(* IEC 61131-3 sources: RL_MAR/experiments/comparison/llm4plc/results/deepseek-ai-DeepSeek-V3.2_20260506_104945/20260506_110433, 4 files *)

(* ---- generated_code_iteration_0.st ---- *)
START_ST
FUNCTION_BLOCK ShellSortFB
VAR_INPUT
    sortDirection : BOOL; // FALSE = ascending, TRUE = descending
    arr : ARRAY[1..1000] OF DINT;
END_VAR
VAR_OUTPUT
    error : BOOL;
    status : WORD;
    sorted_arr : ARRAY[1..1000] OF DINT;
END_VAR
VAR
    state : INT; // 0=INIT, 1=SORTING, 2=COMPLETED, 3=ERROR
    prevState : INT;
    i : DINT;
    j : DINT;
    gap : DINT;
    temp : DINT;
    swapFlag : BOOL;
    N : CONSTANT := 1000;
    internalArray : ARRAY[1..1000] OF DINT;
END_VAR

CASE state OF
    0: // STATE 0: INITIALIZE
        // Copy input array to sorted_arr and internalArray
        FOR i := 1 TO N BY 1 DO
            sorted_arr[i] := arr[i];
            internalArray[i] := arr[i];
        END_FOR;

        // Perform array length validation (N is fixed at 1000)
        IF N <= 1 THEN
            error := TRUE;
            status := 16#8200; // Array size <= 1
            state := 3; // Transition to ERROR state
        ELSIF N > 1000 THEN
            error := TRUE;
            status := 16#8201; // Array size > 1000
            state := 3; // Transition to ERROR state
        ELSE
            error := FALSE;
            status := 16#0000; // No error
            state := 1; // Transition to SORTING state
            gap := N / 2; // Initialize gap for Shell Sort
            swapFlag := FALSE;
        END_IF;

    1: // STATE 1: SORTING
        // Perform Shell Sort algorithm
        IF gap > 0 THEN
            swapFlag := FALSE;
            i := gap + 1;
            WHILE i <= N DO
                temp := internalArray[i];
                j := i;

                // Compare and swap based on sortDirection
                IF NOT sortDirection THEN // Ascending order
                    WHILE (j > gap) AND (internalArray[j - gap] > temp) DO
                        internalArray[j] := internalArray[j - gap];
                        j := j - gap;
                        swapFlag := TRUE;
                    END_WHILE;
                ELSE // Descending order
                    WHILE (j > gap) AND (internalArray[j - gap] < temp) DO
                        internalArray[j] := internalArray[j - gap];
                        j := j - gap;
                        swapFlag := TRUE;
                    END_WHILE;
                END_IF;

                internalArray[j] := temp;
                i := i + 1;
            END_WHILE;

            // Reduce gap if no swaps occurred in this iteration
            IF NOT swapFlag THEN
                gap := gap / 2;
            END_IF;
        ELSE
            // Sorting completed, copy internalArray to sorted_arr
            FOR i := 1 TO N BY 1 DO
                sorted_arr[i] := internalArray[i];
            END_FOR;
            state := 2; // Transition to COMPLETED state
        END_IF;

    2: // STATE 2: COMPLETED
        // Maintain final outputs
        error := FALSE;
        status := 16#0000;
        // sorted_arr already contains sorted result
        // Remain in COMPLETED state
        state := 2;

    3: // STATE 3: ERROR
        // Maintain error outputs
        // sorted_arr already contains copy of input arr (unsorted)
        // Remain in ERROR state
        state := 3;

END_CASE;

prevState := state;
END_FUNCTION_BLOCK
END_ST

(* ---- generated_code_iteration_1.st ---- *)
START_REASON
The validation feedback indicates that the CODESYS compiler validation failed with the message: "应该采用类型定义取代'CONSTANT'". This is Chinese for "should use type definition instead of 'CONSTANT'". In CODESYS Structured Text (IEC 61131-3), the keyword for declaring a constant is `CONSTANT`, but the feedback suggests using a type definition. However, `CONSTANT` is the correct keyword for declaring a constant variable within a VAR section. The issue might be that `CONSTANT` is used in a VAR block where it should be declared differently, or there might be a syntax nuance. In CODESYS, constants in a VAR block are declared with `CONSTANT` after the variable name and type, but the feedback might be pointing to using a type definition (e.g., defining a constant at the global scope) instead. Alternatively, the constant `N` is declared as `N : CONSTANT := 1000;` in the VAR section. According to IEC 61131-3, constants in VAR blocks should be declared as `CONSTANT` with the assignment, but CODESYS might prefer a different syntax or placement. To fix this, I can move the constant declaration to a VAR_CONSTANT section or use a proper type definition. Since the feedback says "type definition", I'll change it to use a VAR_CONSTANT block, which is the standard way to declare constants in a function block. This separates constants from regular variables and should satisfy the CODESYS compiler. I'll restructure the VAR section to include VAR_CONSTANT for N.

Additionally, I'll review the code for other potential issues: The state machine logic and Shell Sort algorithm appear correct, but I'll ensure that the constant is properly defined. The original code uses `N : CONSTANT := 1000;` in VAR, which might be misinterpreted by CODESYS. By moving it to VAR_CONSTANT, I align with best practices.

Let me update the code accordingly.
END_REASON

START_ST
FUNCTION_BLOCK ShellSortFB
VAR_INPUT
    sortDirection : BOOL; // FALSE = ascending, TRUE = descending
    arr : ARRAY[1..1000] OF DINT;
END_VAR
VAR_OUTPUT
    error : BOOL;
    status : WORD;
    sorted_arr : ARRAY[1..1000] OF DINT;
END_VAR
VAR
    state : INT; // 0=INIT, 1=SORTING, 2=COMPLETED, 3=ERROR
    prevState : INT;
    i : DINT;
    j : DINT;
    gap : DINT;
    temp : DINT;
    swapFlag : BOOL;
    internalArray : ARRAY[1..1000] OF DINT;
END_VAR
VAR_CONSTANT
    N : DINT := 1000;
END_VAR

CASE state OF
    0: // STATE 0: INITIALIZE
        // Copy input array to sorted_arr and internalArray
        FOR i := 1 TO N BY 1 DO
            sorted_arr[i] := arr[i];
            internalArray[i] := arr[i];
        END_FOR;

        // Perform array length validation (N is fixed at 1000)
        IF N <= 1 THEN
            error := TRUE;
            status := 16#8200; // Array size <= 1
            state := 3; // Transition to ERROR state
        ELSIF N > 1000 THEN
            error := TRUE;
            status := 16#8201; // Array size > 1000
            state := 3; // Transition to ERROR state
        ELSE
            error := FALSE;
            status := 16#0000; // No error
            state := 1; // Transition to SORTING state
            gap := N / 2; // Initialize gap for Shell Sort
            swapFlag := FALSE;
        END_IF;

    1: // STATE 1: SORTING
        // Perform Shell Sort algorithm
        IF gap > 0 THEN
            swapFlag := FALSE;
            i := gap + 1;
            WHILE i <= N DO
                temp := internalArray[i];
                j := i;

                // Compare and swap based on sortDirection
                IF NOT sortDirection THEN // Ascending order
                    WHILE (j > gap) AND (internalArray[j - gap] > temp) DO
                        internalArray[j] := internalArray[j - gap];
                        j := j - gap;
                        swapFlag := TRUE;
                    END_WHILE;
                ELSE // Descending order
                    WHILE (j > gap) AND (internalArray[j - gap] < temp) DO
                        internalArray[j] := internalArray[j - gap];
                        j := j - gap;
                        swapFlag := TRUE;
                    END_WHILE;
                END_IF;

                internalArray[j] := temp;
                i := i + 1;
            END_WHILE;

            // Reduce gap if no swaps occurred in this iteration
            IF NOT swapFlag THEN
                gap := gap / 2;
            END_IF;
        ELSE
            // Sorting completed, copy internalArray to sorted_arr
            FOR i := 1 TO N BY 1 DO
                sorted_arr[i] := internalArray[i];
            END_FOR;
            state := 2; // Transition to COMPLETED state
        END_IF;

    2: // STATE 2: COMPLETED
        // Maintain final outputs
        error := FALSE;
        status := 16#0000;
        // sorted_arr already contains sorted result
        // Remain in COMPLETED state
        state := 2;

    3: // STATE 3: ERROR
        // Maintain error outputs
        // sorted_arr already contains copy of input arr (unsorted)
        // Remain in ERROR state
        state := 3;

END_CASE;

prevState := state;
END_FUNCTION_BLOCK
END_ST

(* ---- generated_code_iteration_2.st ---- *)
START_REASON
The validation feedback indicates an encoding issue: "ANTLR: ANTLR syntax check failed: 'gbk' codec can't decode byte 0xaf in position 115: illegal multibyte sequence" and similarly for CODESYS. This suggests that the code contains a character that cannot be decoded with the GBK encoding, likely a non-ASCII character. In the previous code, I used Chinese comments (e.g., "FALSE = ascending, TRUE = descending") which might include characters not compatible with GBK or the compiler's expected encoding. The byte 0xaf could correspond to a specific Chinese character or symbol. To fix this, I should remove all non-ASCII characters from the code, including Chinese comments, and replace them with English or simple ASCII text. This ensures compatibility with the compiler's encoding settings.

Additionally, I'll review the code for any other non-ASCII characters. The constant N is defined in VAR_CONSTANT, which should be fine. I'll also ensure that the state machine logic remains correct. The error might also stem from other hidden characters, but removing Chinese comments is the primary step.

Let me update the code by replacing Chinese comments with English equivalents and ensuring all text is ASCII-compatible.
END_REASON

START_ST
FUNCTION_BLOCK ShellSortFB
VAR_INPUT
    sortDirection : BOOL; // FALSE for ascending, TRUE for descending
    arr : ARRAY[1..1000] OF DINT;
END_VAR
VAR_OUTPUT
    error : BOOL;
    status : WORD;
    sorted_arr : ARRAY[1..1000] OF DINT;
END_VAR
VAR
    state : INT; // 0=INIT, 1=SORTING, 2=COMPLETED, 3=ERROR
    prevState : INT;
    i : DINT;
    j : DINT;
    gap : DINT;
    temp : DINT;
    swapFlag : BOOL;
    internalArray : ARRAY[1..1000] OF DINT;
END_VAR
VAR_CONSTANT
    N : DINT := 1000;
END_VAR

CASE state OF
    0: // STATE 0: INITIALIZE
        // Copy input array to sorted_arr and internalArray
        FOR i := 1 TO N BY 1 DO
            sorted_arr[i] := arr[i];
            internalArray[i] = arr[i];
        END_FOR;

        // Perform array length validation (N is fixed at 1000)
        IF N <= 1 THEN
            error := TRUE;
            status := 16#8200; // Array size <= 1 error
            state := 3; // Transition to ERROR state
        ELSIF N > 1000 THEN
            error := TRUE;
            status := 16#8201; // Array size > 1000 error
            state := 3; // Transition to ERROR state
        ELSE
            error := FALSE;
            status := 16#0000; // No error
            state := 1; // Transition to SORTING state
            gap := N / 2; // Initialize gap for Shell Sort
            swapFlag := FALSE;
        END_IF;

    1: // STATE 1: SORTING
        // Perform Shell Sort algorithm
        IF gap > 0 THEN
            swapFlag := FALSE;
            i := gap + 1;
            WHILE i <= N DO
                temp := internalArray[i];
                j := i;

                // Compare and swap based on sortDirection
                IF NOT sortDirection THEN // Ascending order
                    WHILE (j > gap) AND (internalArray[j - gap] > temp) DO
                        internalArray[j] := internalArray[j - gap];
                        j := j - gap;
                        swapFlag := TRUE;
                    END_WHILE;
                ELSE // Descending order
                    WHILE (j > gap) AND (internalArray[j - gap] < temp) DO
                        internalArray[j] := internalArray[j - gap];
                        j := j - gap;
                        swapFlag := TRUE;
                    END_WHILE;
                END_IF;

                internalArray[j] := temp;
                i := i + 1;
            END_WHILE;

            // Reduce gap if no swaps occurred in this iteration
            IF NOT swapFlag THEN
                gap := gap / 2;
            END_IF;
        ELSE
            // Sorting completed, copy internalArray to sorted_arr
            FOR i := 1 TO N BY 1 DO
                sorted_arr[i] := internalArray[i];
            END_FOR;
            state := 2; // Transition to COMPLETED state
        END_IF;

    2: // STATE 2: COMPLETED
        // Maintain final outputs
        error := FALSE;
        status := 16#0000;
        // sorted_arr already contains sorted result
        // Remain in COMPLETED state
        state := 2;

    3: // STATE 3: ERROR
        // Maintain error outputs
        // sorted_arr already contains copy of input arr (unsorted)
        // Remain in ERROR state
        state := 3;

END_CASE;

prevState := state;
END_FUNCTION_BLOCK
END_ST

(* ---- generated_code_iteration_3.st ---- *)
START_REASON
The CODESYS compiler validation error indicates that "VAR_CONSTANT" is not allowed in the current context. In CODESYS Structured Text, constants should be defined within the VAR section using the "CONSTANT" keyword, not in a separate VAR_CONSTANT block. The error message specifically says: "应该采用VAR, VAR_INPUT, VAR_OUTPUT 或 VAR_IN_OUT 取代VAR_CONSTANT", which translates to "Should use VAR, VAR_INPUT, VAR_OUTPUT or VAR_IN_OUT instead of VAR_CONSTANT".

I need to move the constant definition from VAR_CONSTANT to the VAR section with the CONSTANT keyword. The constant N should be declared as:
VAR CONSTANT
    N : DINT := 1000;
END_VAR

This is the proper way to define constants in CODESYS Structured Text. I'll make this change while keeping all other code structure the same.
END_REASON

START_ST
FUNCTION_BLOCK ShellSortFB
VAR_INPUT
    sortDirection : BOOL; // FALSE for ascending, TRUE for descending
    arr : ARRAY[1..1000] OF DINT;
END_VAR
VAR_OUTPUT
    error : BOOL;
    status : WORD;
    sorted_arr : ARRAY[1..1000] OF DINT;
END_VAR
VAR
    state : INT; // 0=INIT, 1=SORTING, 2=COMPLETED, 3=ERROR
    prevState : INT;
    i : DINT;
    j : DINT;
    gap : DINT;
    temp : DINT;
    swapFlag : BOOL;
    internalArray : ARRAY[1..1000] OF DINT;
END_VAR
VAR CONSTANT
    N : DINT := 1000;
END_VAR

CASE state OF
    0: // STATE 0: INITIALIZE
        // Copy input array to sorted_arr and internalArray
        FOR i := 1 TO N BY 1 DO
            sorted_arr[i] := arr[i];
            internalArray[i] := arr[i];
        END_FOR;

        // Perform array length validation (N is fixed at 1000)
        IF N <= 1 THEN
            error := TRUE;
            status := 16#8200; // Array size <= 1 error
            state := 3; // Transition to ERROR state
        ELSIF N > 1000 THEN
            error := TRUE;
            status := 16#8201; // Array size > 1000 error
            state := 3; // Transition to ERROR state
        ELSE
            error := FALSE;
            status := 16#0000; // No error
            state := 1; // Transition to SORTING state
            gap := N / 2; // Initialize gap for Shell Sort
            swapFlag := FALSE;
        END_IF;

    1: // STATE 1: SORTING
        // Perform Shell Sort algorithm
        IF gap > 0 THEN
            swapFlag := FALSE;
            i := gap + 1;
            WHILE i <= N DO
                temp := internalArray[i];
                j := i;

                // Compare and swap based on sortDirection
                IF NOT sortDirection THEN // Ascending order
                    WHILE (j > gap) AND (internalArray[j - gap] > temp) DO
                        internalArray[j] := internalArray[j - gap];
                        j := j - gap;
                        swapFlag := TRUE;
                    END_WHILE;
                ELSE // Descending order
                    WHILE (j > gap) AND (internalArray[j - gap] < temp) DO
                        internalArray[j] := internalArray[j - gap];
                        j := j - gap;
                        swapFlag := TRUE;
                    END_WHILE;
                END_IF;

                internalArray[j] := temp;
                i := i + 1;
            END_WHILE;

            // Reduce gap if no swaps occurred in this iteration
            IF NOT swapFlag THEN
                gap := gap / 2;
            END_IF;
        ELSE
            // Sorting completed, copy internalArray to sorted_arr
            FOR i := 1 TO N BY 1 DO
                sorted_arr[i] := internalArray[i];
            END_FOR;
            state := 2; // Transition to COMPLETED state
        END_IF;

    2: // STATE 2: COMPLETED
        // Maintain final outputs
        error := FALSE;
        status := 16#0000;
        // sorted_arr already contains sorted result
        // Remain in COMPLETED state
        state := 2;

    3: // STATE 3: ERROR
        // Maintain error outputs
        // sorted_arr already contains copy of input arr (unsorted)
        // Remain in ERROR state
        state := 3;

END_CASE;

prevState := state;
END_FUNCTION_BLOCK
END_ST
